// TIA Portal V18 export
DATA_BLOCK "SqlCommands"   // DB3
TITLE = SqlCommands
{ S7_Optimized_Access := 'TRUE' }
AUTHOR : SIEMENS SUP Applications
VERSION : 1.1
// DB for holding the command strings for a Tabular Data Stream command to a SQL database
// stored: MemoryReserve 0
   VAR
      currentSqlCommand { ExternalAccessible := 'False'; ExternalVisible := 'False'; ExternalWritable := 'False'} : USInt := 6;   // index of current SQL command to be executed (zero-based)
      sqlCommands { ExternalAccessible := 'False'; ExternalVisible := 'False'; ExternalWritable := 'False'} : Array[0..25] of String;   // array of SQL command strings
   END_VAR
BEGIN
   sqlCommands[0] := 'insert into PLCDATA_1 values (7,8, 9)';
   sqlCommands[1] := 'Update PLCDATA_1 set IntegerValue1 = 7, IntegerValue2 = 7, IntegerValue3 = 7 where IntegerValue2 = 7';
   sqlCommands[2] := 'Select IntegerValue1 from PLCDATA_1';
   sqlCommands[3] := 'Select Fruit from PLCDATA_2 where Amount != 0';
   sqlCommands[4] := 'Select Fruit from PLCDATA_2 where color = $'red$'';
   sqlCommands[5] := 'insert into PLCDATA_3 values (7, $'2020-01-01 10:23:24.125$')';
   sqlCommands[6] := 'SELECT TOP (3) * FROM PLCDATA ORDER BY Temperature';
   sqlCommands[7] := 'execute myProcedureIn @input1=30, @input2=6, @input3=84';
   sqlCommands[8] := 'execute myProcedureSelect';
   sqlCommands[9] := 'declare @myout1 char(30),  @myout2 int execute myProcedureInOut @in1=$'pear$', @in2=$'yellow$', @in3=3, @out1=@myout1 OUTPUT, @out2=@myout2 OUTPUT select @myout1 as $'myOut1$', @myOut2 as $'myOut2$'';
   sqlCommands[10] := 'INSERT INTO [dbo].[errors] ([Text]) VALUES ($'remotetest$')';
   sqlCommands[11] := 'SELECT TOP (10) ValueReal1, ValueReal2, ValueReal3, ValueReal4, ValueReal5, ValueReal6, ValueReal7, ValueReal8, ValueReal9 FROM TestJulian';
   sqlCommands[12] := 'SELECT * FROM KompressionLog ORDER BY StentNr';
   sqlCommands[13] := 'execute SelectProc1';
   sqlCommands[14] := 'insert into TestDateTime values ($'01.01.1990 12:00:00$')';
   sqlCommands[15] := 'exec SetDateTime @Input1 = $'07.30.1990 12:00:00$'';
   sqlCommands[16] := 'SELECT TOP (100) MesId, MesId2, MesId3 FROM TestJulian';
   sqlCommands[17] := 'SELECT TOP (1) DateTime FROM TestDateTime';
   sqlCommands[18] := 'SELECT TOP 2 * FROM FunctionTest ORDER BY ID';
   sqlCommands[19] := 'INSERT INTO [dbo].[FunctionTest] DEFAULT VALUES';
   sqlCommands[20] := 'use [SQLFromPLC] declare @myout1 bit  execute  NachtragDatensaetze @inDateiPfad= $'C:\Program Files\Microsoft SQL Server\MSSQL14.SQLEXPRESS\MSSQL\DATA\iO.csv$', @outDone=@myout1 OUTPUT select @myout1 as $'myOut1$'';
   sqlCommands[21] := 'UPDATE [dbo].[KompressionLog] SET LotNummer = $'Test234$' WHERE KammerId = $'3$'';
END_DATA_BLOCK
